FUNCTION F_SetExternalFunctionError : BOOL
(**************************************************************************************
 * 	Application		:	BoxControl Framework
 *	Revision		:	$Revision: 404529 $
 *	Revision date	:	$Date: 2018-04-23 08:21:38 +0200 (Mo., 23 Apr 2018) $
 *	Last changed by	:	$Author: b7bolm $
 *	URL				:	$URL: http://almscdc.swisslog.com/repo/SWPD/Development/BoxControlFramework/20_Release/trunk/01_Software/BCF/BCF/JumpStart/20_Product/10_App/12_E_Functions/10_Lib/10_Conv/10_Functions/F_SetExternalFunctionError.TcPOU $
 *
 *	Purpose			:	Set external error
 *						Add an External error, which will be reported over the configured
 *						position.
 *						
 *
 * ------------------------------------------------------------------------------------
 *	Copyright Swisslog [IP AG], Switzerland. All rights reserved.
 * 
 * ------------------------------------------------------------------------------------
 *	
 * 	Revision History: 
 *
 * 	VERSION			DATE			INITIALS			DESCRIPTION
 *	0.1				01.01.2001		swl					Example
 *
 **************************************************************************************)
VAR_INPUT
	eFunctionNumber : E_FunctionNumber; 
	ZoneNumber		: INT;
	ErrorType		: E_ErrorType; // Error message type
	ErrorParam		: STRING(System.ERROR_PARAM_STRINGLENGTH); // Error parameter
	ErrorMsg		: INT; // Error message as String (Will be mapped to error code)
END_VAR


// Validate inputs
IF eFunctionNumber > E_FunctionNumber.F_BEGIN_FUNCTION THEN
	IF __ISVALIDREF(FunctionRegistry[eFunctionNumber].rFunction) THEN
		// Set external error on instance
		FunctionRegistry[eFunctionNumber].rFunction.M_SetExternalError(
			mZoneNumber := ZoneNumber,
			mErrorType 	:= ErrorType,
			mErrorParam := ErrorParam,
			mErrorCode 	:= ErrorMsg);
	END_IF
END_IF

END_FUNCTION

(* stored: Version 1.1.0.1, ProductVersion 3.1.4022.12
   POU F_SetExternalFunctionError: Id {cecf8fcc-6b8f-4290-8d08-b033c92ce7f4}, SpecialFunc None *)
